(* Logix 5000 project; controller PLC vendor 1 type 14 code 155 rev 30.14; software revision 30.01; part 3 of 4 *)
(* tags used below, declared in another part *)
   Alarm_Word_Current : DINT[3];
   Bridge_Timer_Gearing_Delay : TIMER;
   Bridge_Timer_Gearing_Delay_DN_OS : BOOL;
   Depositor : Depositor_R2b;
   Encoder_Conveyor : AXIS_CIP_DRIVE;
   FORCE_GO_SIGNAL : BOOL;
   Forces : Forces_R2b;
   homing_timeout : TIMER;
   IO : IO_R2a;
   MV_conveyor_stopped : BOOL;
   MV_Encoder_Stop_Value : REAL;
   mv_index_counter : COUNTER;
   MV_indexes : DINT;
   MV_total_indexes : COUNTER;
   OS : INT[10];
   Recipe_Setpoints_DINT : DINT[23,20];
   Sequencer_Auto : Sequencer_R2a;
   Sequencer_Home : Sequencer_R2a;
   Servo_Bridge_Shift : AXIS_CIP_DRIVE;
   Servo_MC_Bridge_Shift : Axis_MC_R3b;
   System : System_R2e;
   Test_Bits : BOOL[32];
   Timers : TIMER[20];   // x
(* MainProgram, continued *)

ROUTINE File_012_Digital_Outputs   (* ladder *)
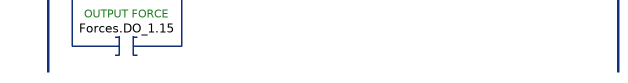
   // DIGITAL OUTPUT MAPPING
   0: [[XIC(IO.DO_1.0) ,XIC(Forces.DO_1.0) ] OTE(Local:1:O.Data.0) ,[XIC(IO.DO_1.1) ,XIC(Forces.DO_1.1) ] OTE(Local:1:O.Data.1) ,[XIC(IO.DO_1.2) ,XIC(Forces.DO_1.2) ] OTE(Local:1:O.Data.2) ,[XIC(IO.DO_1.3) ,XIC(Forces.DO_1.3) ] OTE(Local:1:O.Data.3) ,[XIC(IO.DO_1.4) ,XIC(Forces.DO_1.4) ] OTE(Local:1:O.Data.4) ,[XIC(IO.DO_1.5) ,XIC(Forces.DO_1.5) ] OTE(Local:1:O.Data.5) ,[XIC(IO.DO_1.6) ,XIC(Forces.DO_1.6) ] OTE(Local:1:O.Data.6) ,[XIC(IO.DO_1.7) ,XIC(Forces.DO_1.7) ] OTE(Local:1:O.Data.7) ,[XIC(IO.DO_1.8) ,XIC(Forces.DO_1.8) ] OTE(Local:1:O.Data.8) ,[XIC(IO.DO_1.9) ,XIC(Forces.DO_1.9) ] OTE(Local:1:O.Data.9) ,[XIC(IO.DO_1.10) ,XIC(Forces.DO_1.10) ] OTE(Local:1:O.Data.10) ,[XIC(IO.DO_1.11) ,XIC(Forces.DO_1.11) ] OTE(Local:1:O.Data.11) ,[XIC(IO.DO_1.12) ,XIC(Forces.DO_1.12) ] OTE(Local:1:O.Data.12) ,[XIC(IO.DO_1.13) ,XIC(Forces.DO_1.13) ] OTE(Local:1:O.Data.13) ,[XIC(IO.DO_1.14) ,XIC(Forces.DO_1.14) ] OTE(Local:1:O.Data.14) ,[XIC(IO.DO_1.15) ,XIC(Forces.DO_1.15) ] OTE(Local:1:O.Data.15) ];
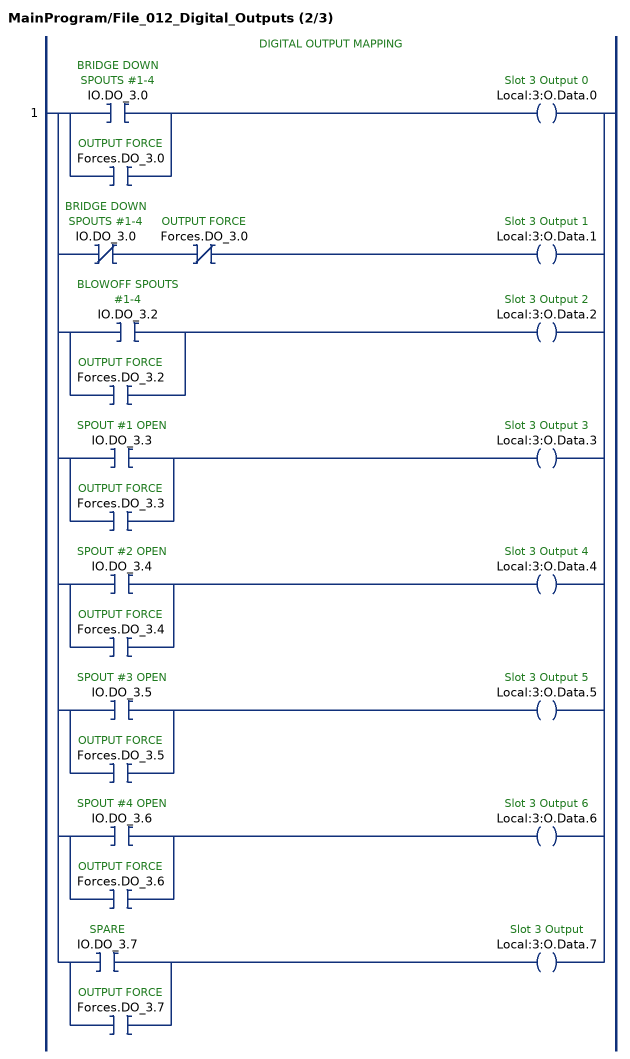
   // DIGITAL OUTPUT MAPPING
   1: [[XIC(IO.DO_3.0) ,XIC(Forces.DO_3.0) ] OTE(Local:3:O.Data.0) ,XIO(IO.DO_3.0) XIO(Forces.DO_3.0) OTE(Local:3:O.Data.1) ,[XIC(IO.DO_3.2) ,XIC(Forces.DO_3.2) ] OTE(Local:3:O.Data.2) ,[XIC(IO.DO_3.3) ,XIC(Forces.DO_3.3) ] OTE(Local:3:O.Data.3) ,[XIC(IO.DO_3.4) ,XIC(Forces.DO_3.4) ] OTE(Local:3:O.Data.4) ,[XIC(IO.DO_3.5) ,XIC(Forces.DO_3.5) ] OTE(Local:3:O.Data.5) ,[XIC(IO.DO_3.6) ,XIC(Forces.DO_3.6) ] OTE(Local:3:O.Data.6) ,[XIC(IO.DO_3.7) ,XIC(Forces.DO_3.7) ] OTE(Local:3:O.Data.7) ];
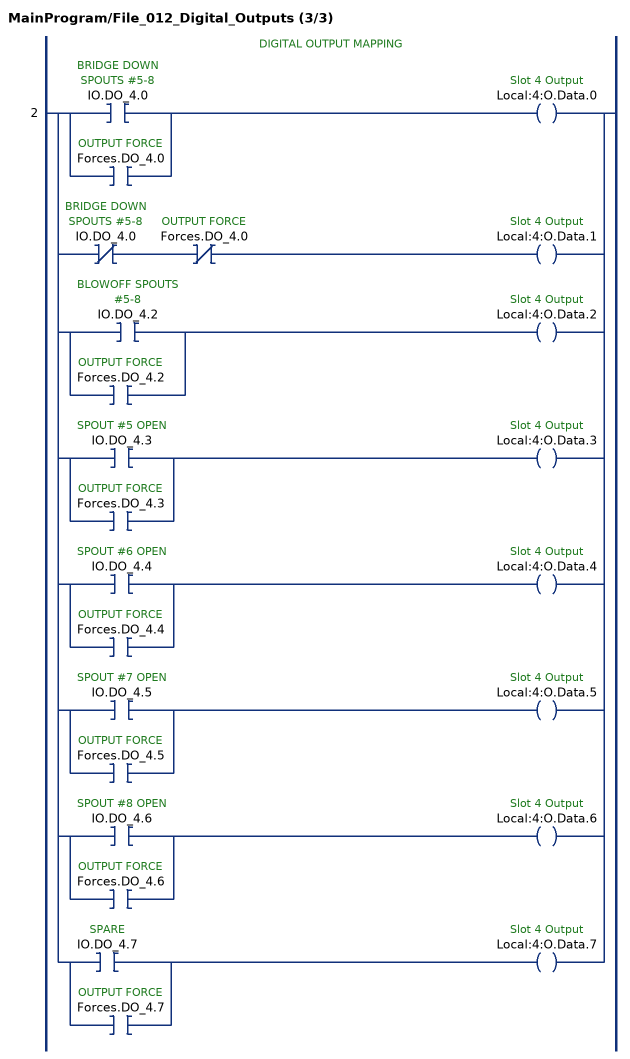
   // DIGITAL OUTPUT MAPPING
   2: [[XIC(IO.DO_4.0) ,XIC(Forces.DO_4.0) ] OTE(Local:4:O.Data.0) ,XIO(IO.DO_4.0) XIO(Forces.DO_4.0) OTE(Local:4:O.Data.1) ,[XIC(IO.DO_4.2) ,XIC(Forces.DO_4.2) ] OTE(Local:4:O.Data.2) ,[XIC(IO.DO_4.3) ,XIC(Forces.DO_4.3) ] OTE(Local:4:O.Data.3) ,[XIC(IO.DO_4.4) ,XIC(Forces.DO_4.4) ] OTE(Local:4:O.Data.4) ,[XIC(IO.DO_4.5) ,XIC(Forces.DO_4.5) ] OTE(Local:4:O.Data.5) ,[XIC(IO.DO_4.6) ,XIC(Forces.DO_4.6) ] OTE(Local:4:O.Data.6) ,[XIC(IO.DO_4.7) ,XIC(Forces.DO_4.7) ] OTE(Local:4:O.Data.7) ];
END_ROUTINE

ROUTINE File_030_Sequencer_Homing   (* ladder *)
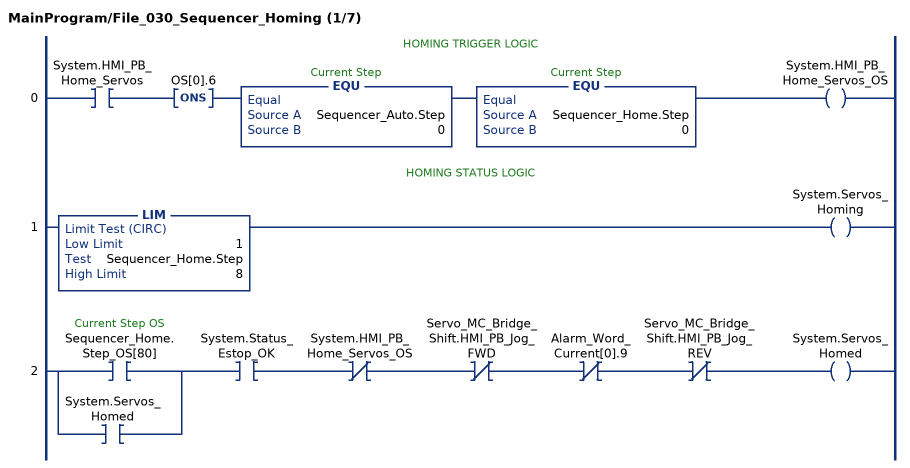
   // HOMING TRIGGER LOGIC
   0: XIC(System.HMI_PB_Home_Servos)ONS(OS[0].6)EQU(Sequencer_Auto.Step,0)EQU(Sequencer_Home.Step,0)OTE(System.HMI_PB_Home_Servos_OS);
   // HOMING STATUS LOGIC
   1: LIM(1,Sequencer_Home.Step,8)OTE(System.Servos_Homing);
   2: [XIC(Sequencer_Home.Step_OS[80]) ,XIC(System.Servos_Homed) ]XIC(System.Status_Estop_OK)XIO(System.HMI_PB_Home_Servos_OS)XIO(Servo_MC_Bridge_Shift.HMI_PB_Jog_FWD)XIO(Alarm_Word_Current[0].9)XIO(Servo_MC_Bridge_Shift.HMI_PB_Jog_REV)OTE(System.Servos_Homed);
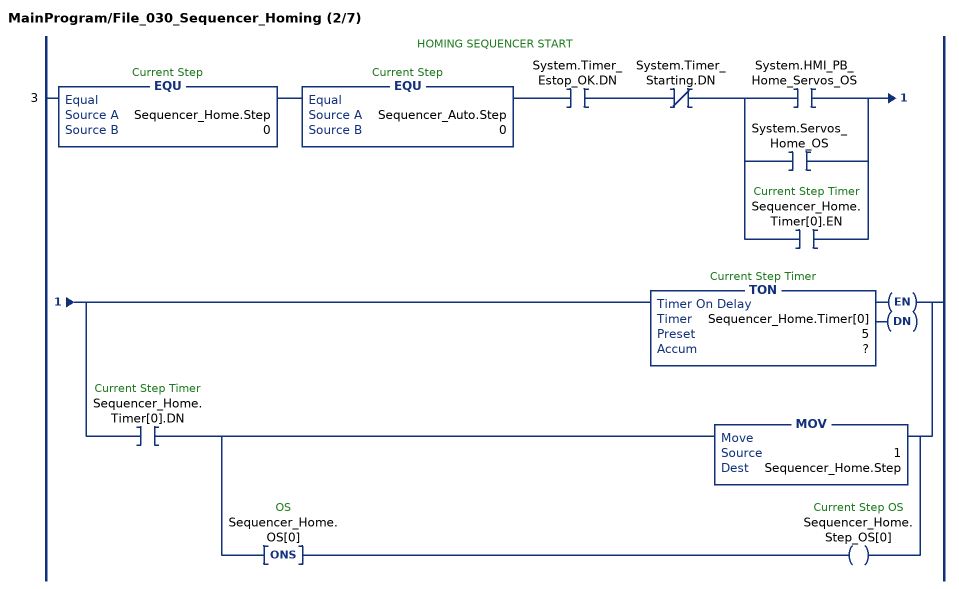
   // HOMING SEQUENCER START
   3: EQU(Sequencer_Home.Step,0)EQU(Sequencer_Auto.Step,0)XIC(System.Timer_Estop_OK.DN)XIO(System.Timer_Starting.DN)[XIC(System.HMI_PB_Home_Servos_OS) ,XIC(System.Servos_Home_OS) ,XIC(Sequencer_Home.Timer[0].EN) ][TON(Sequencer_Home.Timer[0],?,?) ,XIC(Sequencer_Home.Timer[0].DN) [MOV(1,Sequencer_Home.Step) ,ONS(Sequencer_Home.OS[0]) OTE(Sequencer_Home.Step_OS[0]) ] ];
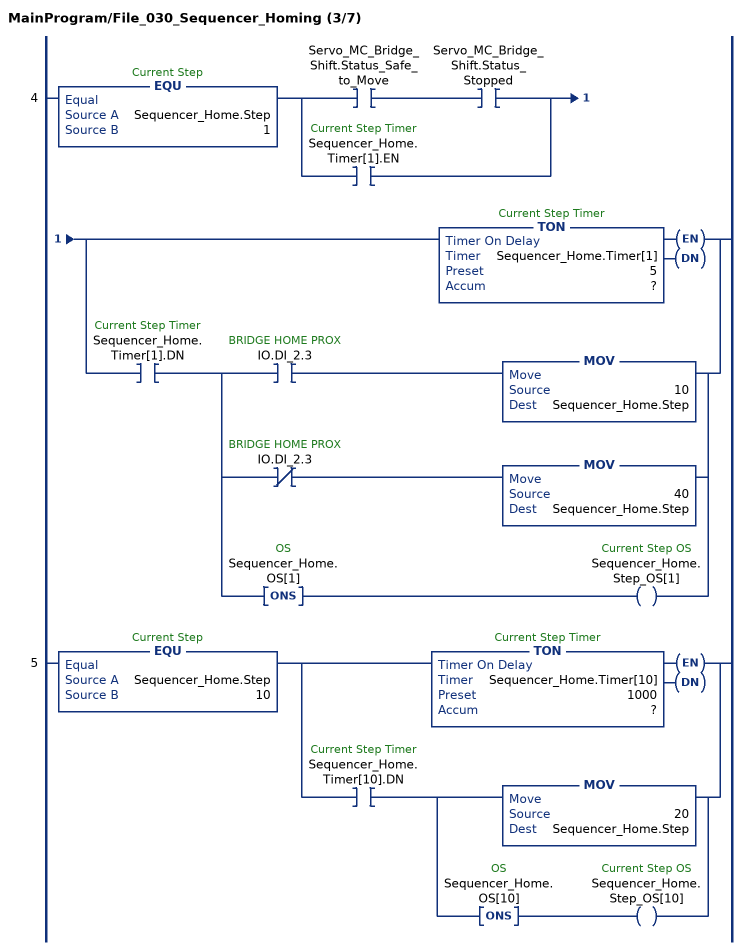
   4: EQU(Sequencer_Home.Step,1)[XIC(Servo_MC_Bridge_Shift.Status_Safe_to_Move) XIC(Servo_MC_Bridge_Shift.Status_Stopped) ,XIC(Sequencer_Home.Timer[1].EN) ][TON(Sequencer_Home.Timer[1],?,?) ,XIC(Sequencer_Home.Timer[1].DN) [XIC(IO.DI_2.3) MOV(10,Sequencer_Home.Step) ,XIO(IO.DI_2.3) MOV(40,Sequencer_Home.Step) ,ONS(Sequencer_Home.OS[1]) OTE(Sequencer_Home.Step_OS[1]) ] ];
   5: EQU(Sequencer_Home.Step,10)[TON(Sequencer_Home.Timer[10],?,?) ,XIC(Sequencer_Home.Timer[10].DN) [MOV(20,Sequencer_Home.Step) ,ONS(Sequencer_Home.OS[10]) OTE(Sequencer_Home.Step_OS[10]) ] ];
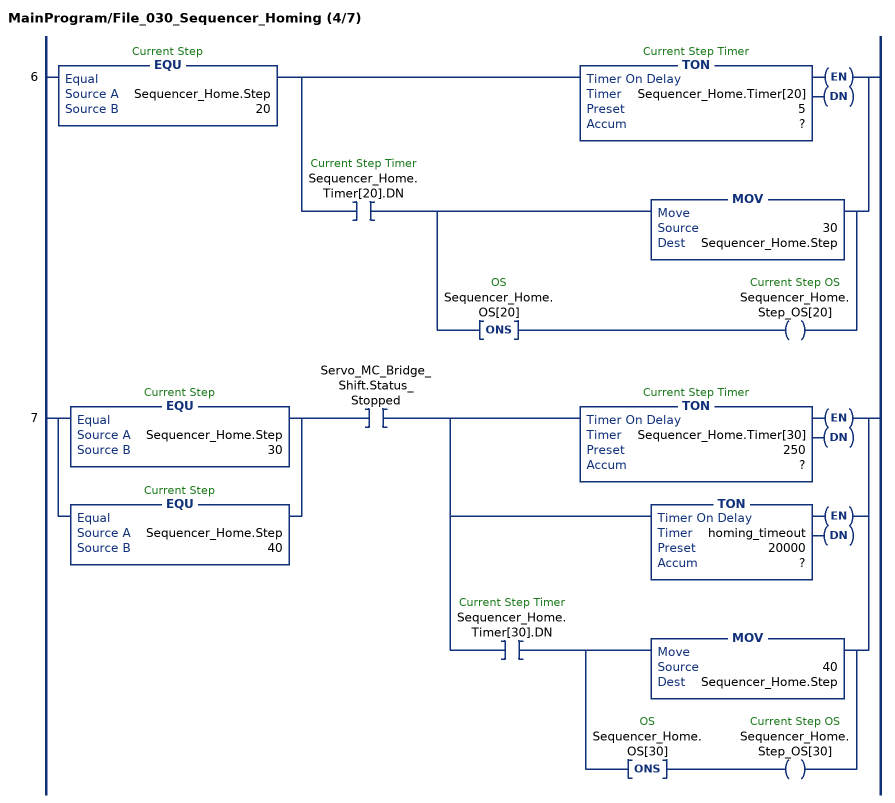
   6: EQU(Sequencer_Home.Step,20)[TON(Sequencer_Home.Timer[20],?,?) ,XIC(Sequencer_Home.Timer[20].DN) [MOV(30,Sequencer_Home.Step) ,ONS(Sequencer_Home.OS[20]) OTE(Sequencer_Home.Step_OS[20]) ] ];
   7: [EQU(Sequencer_Home.Step,30) ,EQU(Sequencer_Home.Step,40) ]XIC(Servo_MC_Bridge_Shift.Status_Stopped)[[TON(Sequencer_Home.Timer[30],?,?) ,TON(homing_timeout,?,?) ] ,XIC(Sequencer_Home.Timer[30].DN) [MOV(40,Sequencer_Home.Step) ,ONS(Sequencer_Home.OS[30]) OTE(Sequencer_Home.Step_OS[30]) ] ];
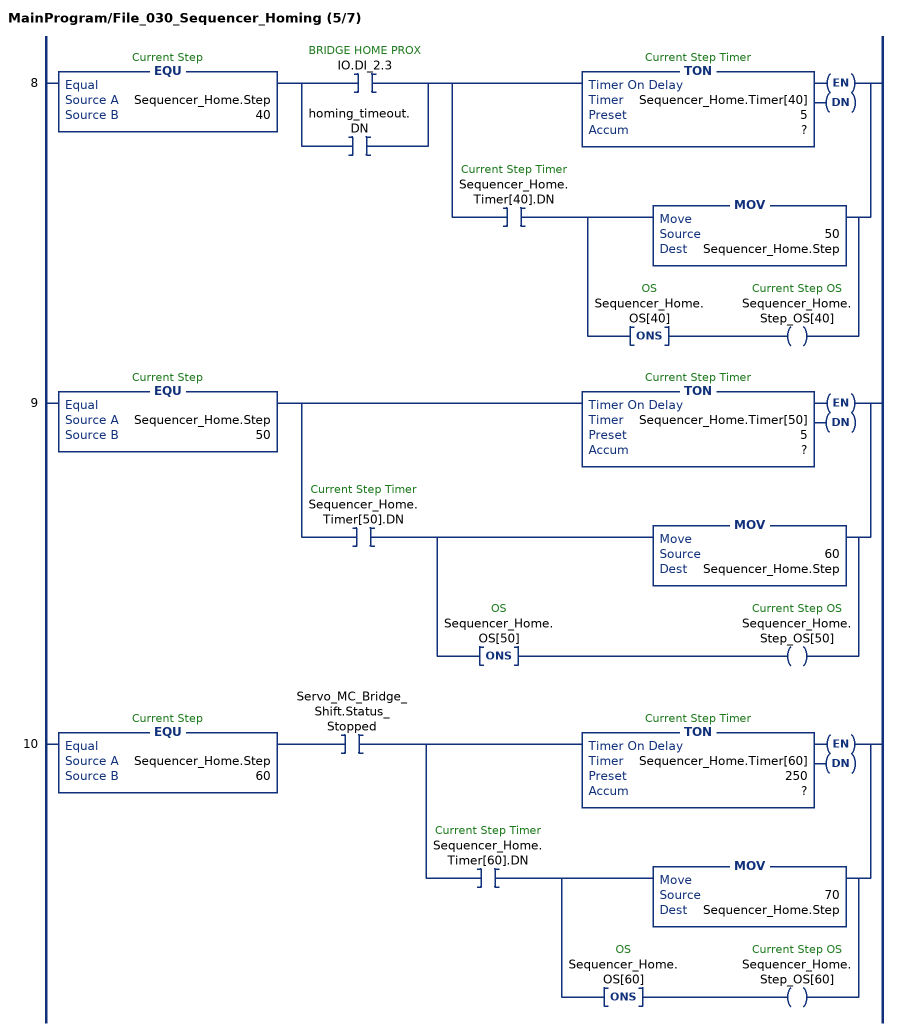
   8: EQU(Sequencer_Home.Step,40)[XIC(IO.DI_2.3) ,XIC(homing_timeout.DN) ][TON(Sequencer_Home.Timer[40],?,?) ,XIC(Sequencer_Home.Timer[40].DN) [MOV(50,Sequencer_Home.Step) ,ONS(Sequencer_Home.OS[40]) OTE(Sequencer_Home.Step_OS[40]) ] ];
   9: EQU(Sequencer_Home.Step,50)[TON(Sequencer_Home.Timer[50],?,?) ,XIC(Sequencer_Home.Timer[50].DN) [MOV(60,Sequencer_Home.Step) ,ONS(Sequencer_Home.OS[50]) OTE(Sequencer_Home.Step_OS[50]) ] ];
   10: EQU(Sequencer_Home.Step,60)XIC(Servo_MC_Bridge_Shift.Status_Stopped)[TON(Sequencer_Home.Timer[60],?,?) ,XIC(Sequencer_Home.Timer[60].DN) [MOV(70,Sequencer_Home.Step) ,ONS(Sequencer_Home.OS[60]) OTE(Sequencer_Home.Step_OS[60]) ] ];
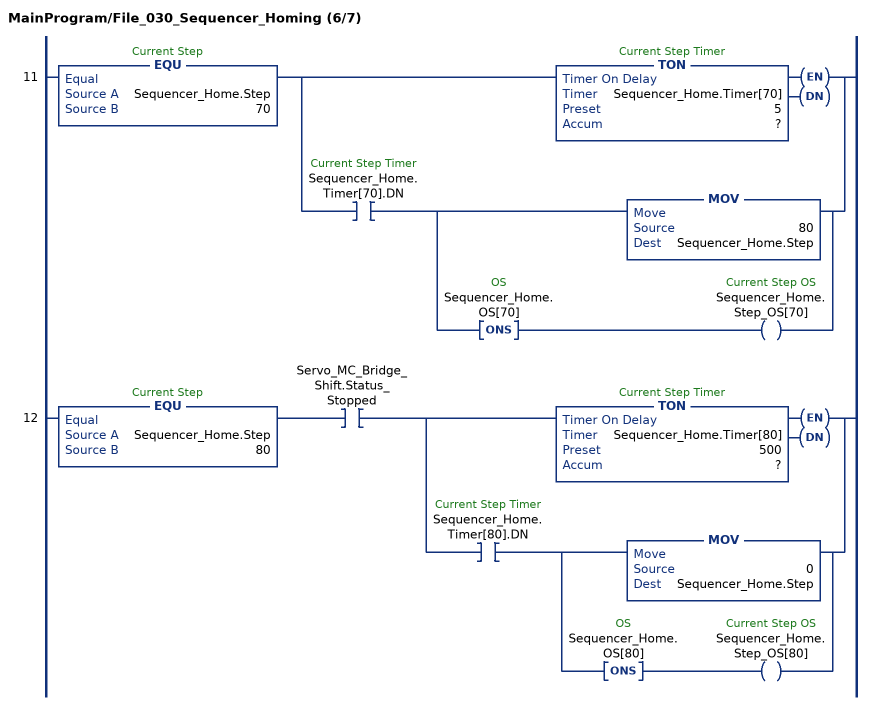
   11: EQU(Sequencer_Home.Step,70)[TON(Sequencer_Home.Timer[70],?,?) ,XIC(Sequencer_Home.Timer[70].DN) [MOV(80,Sequencer_Home.Step) ,ONS(Sequencer_Home.OS[70]) OTE(Sequencer_Home.Step_OS[70]) ] ];
   12: EQU(Sequencer_Home.Step,80)XIC(Servo_MC_Bridge_Shift.Status_Stopped)[TON(Sequencer_Home.Timer[80],?,?) ,XIC(Sequencer_Home.Timer[80].DN) [MOV(0,Sequencer_Home.Step) ,ONS(Sequencer_Home.OS[80]) OTE(Sequencer_Home.Step_OS[80]) ] ];
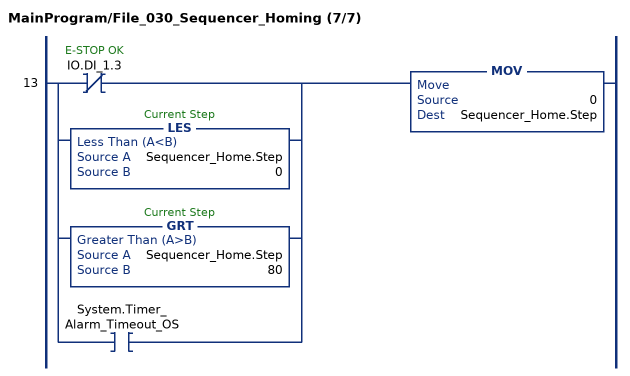
   13: [XIO(IO.DI_1.3) ,LES(Sequencer_Home.Step,0) ,GRT(Sequencer_Home.Step,80) ,XIC(System.Timer_Alarm_Timeout_OS) ]MOV(0,Sequencer_Home.Step);
END_ROUTINE

ROUTINE File_040_Sequencer_Auto   (* ladder *)
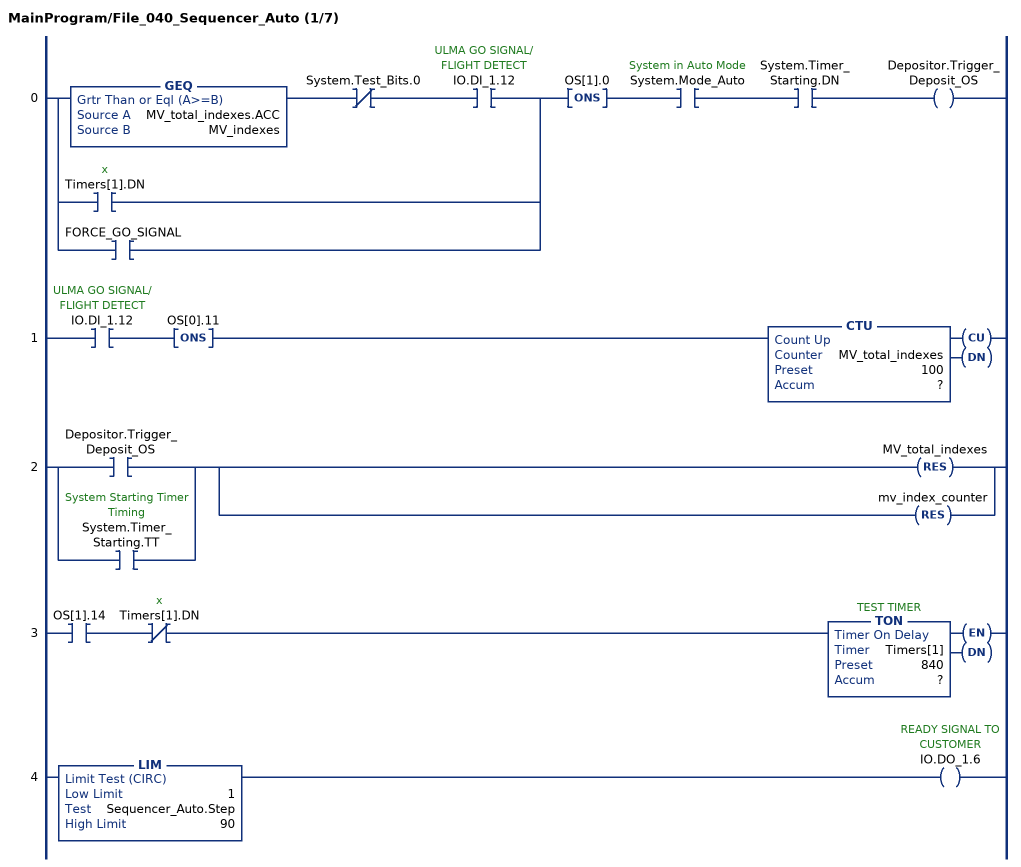
   0: [GEQ(MV_total_indexes.ACC,MV_indexes) XIO(System.Test_Bits.0) XIC(IO.DI_1.12) ,XIC(Timers[1].DN) ,XIC(FORCE_GO_SIGNAL) ]ONS(OS[1].0)XIC(System.Mode_Auto)XIC(System.Timer_Starting.DN)OTE(Depositor.Trigger_Deposit_OS);
   1: XIC(IO.DI_1.12)ONS(OS[0].11)CTU(MV_total_indexes,?,?);
   2: [XIC(Depositor.Trigger_Deposit_OS) ,XIC(System.Timer_Starting.TT) ][RES(MV_total_indexes) ,RES(mv_index_counter) ];
   3: XIC(OS[1].14)XIO(Timers[1].DN)TON(Timers[1],?,?);
   4: LIM(1,Sequencer_Auto.Step,90)OTE(IO.DO_1.6);
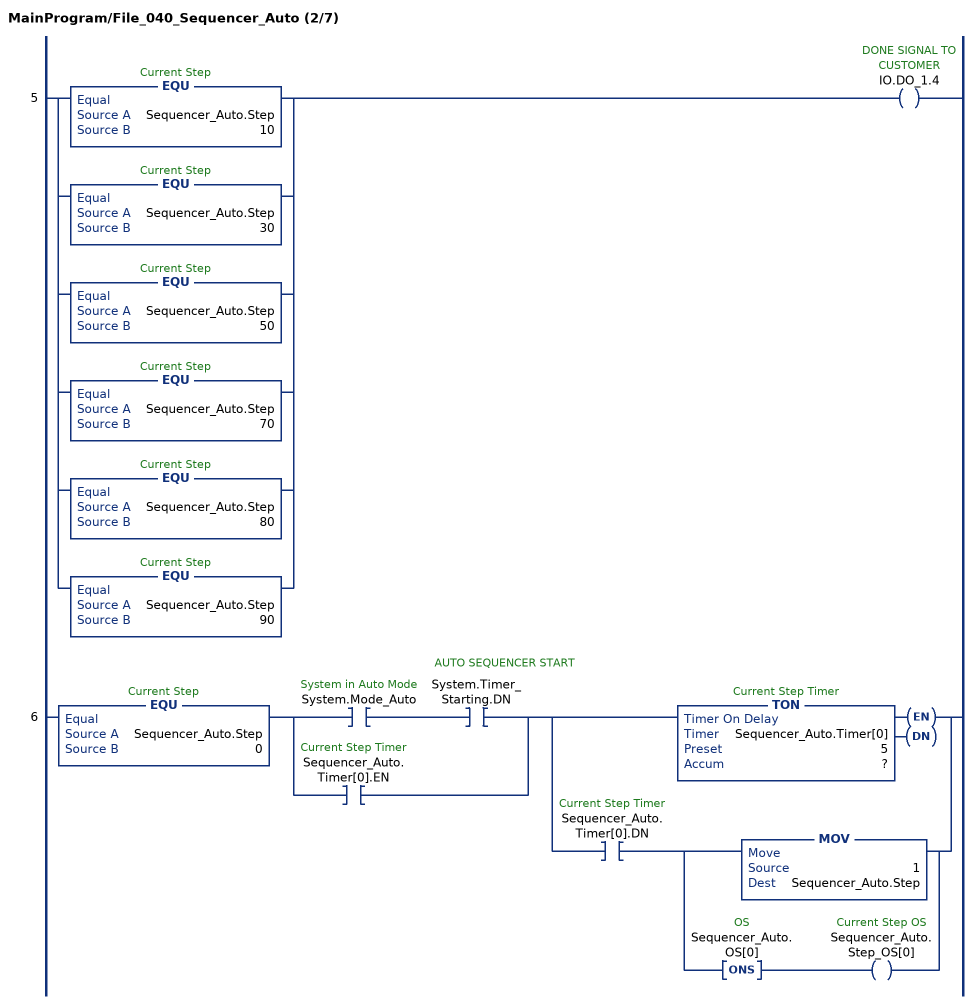
   5: [EQU(Sequencer_Auto.Step,10) ,EQU(Sequencer_Auto.Step,30) ,EQU(Sequencer_Auto.Step,50) ,EQU(Sequencer_Auto.Step,70) ,EQU(Sequencer_Auto.Step,80) ,EQU(Sequencer_Auto.Step,90) ]OTE(IO.DO_1.4);
   // AUTO SEQUENCER START
   6: EQU(Sequencer_Auto.Step,0)[XIC(System.Mode_Auto) XIC(System.Timer_Starting.DN) ,XIC(Sequencer_Auto.Timer[0].EN) ][TON(Sequencer_Auto.Timer[0],?,?) ,XIC(Sequencer_Auto.Timer[0].DN) [MOV(1,Sequencer_Auto.Step) ,ONS(Sequencer_Auto.OS[0]) OTE(Sequencer_Auto.Step_OS[0]) ] ];
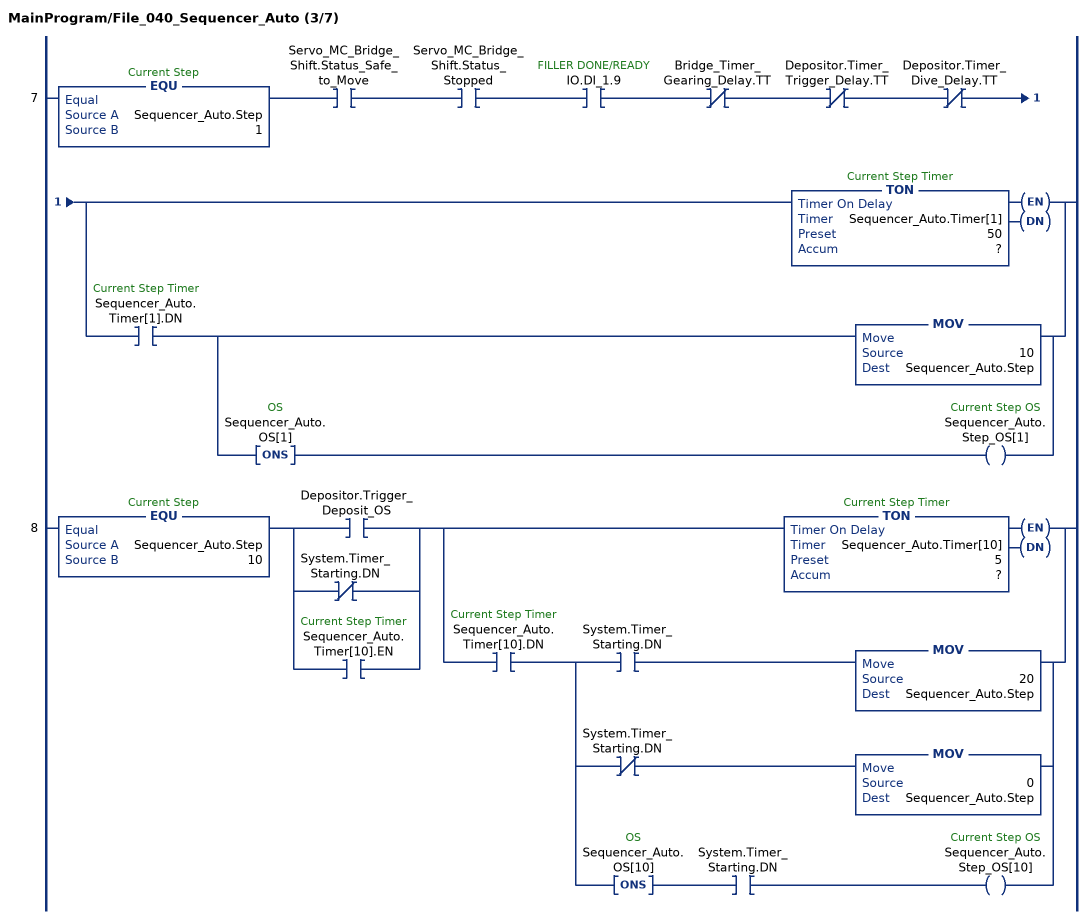
   7: EQU(Sequencer_Auto.Step,1)XIC(Servo_MC_Bridge_Shift.Status_Safe_to_Move)XIC(Servo_MC_Bridge_Shift.Status_Stopped)XIC(IO.DI_1.9)XIO(Bridge_Timer_Gearing_Delay.TT)XIO(Depositor.Timer_Trigger_Delay.TT)XIO(Depositor.Timer_Dive_Delay.TT)[TON(Sequencer_Auto.Timer[1],?,?) ,XIC(Sequencer_Auto.Timer[1].DN) [MOV(10,Sequencer_Auto.Step) ,ONS(Sequencer_Auto.OS[1]) OTE(Sequencer_Auto.Step_OS[1]) ] ];
   8: EQU(Sequencer_Auto.Step,10)[XIC(Depositor.Trigger_Deposit_OS) ,XIO(System.Timer_Starting.DN) ,XIC(Sequencer_Auto.Timer[10].EN) ][TON(Sequencer_Auto.Timer[10],?,?) ,XIC(Sequencer_Auto.Timer[10].DN) [XIC(System.Timer_Starting.DN) MOV(20,Sequencer_Auto.Step) ,XIO(System.Timer_Starting.DN) MOV(0,Sequencer_Auto.Step) ,ONS(Sequencer_Auto.OS[10]) XIC(System.Timer_Starting.DN) OTE(Sequencer_Auto.Step_OS[10]) ] ];
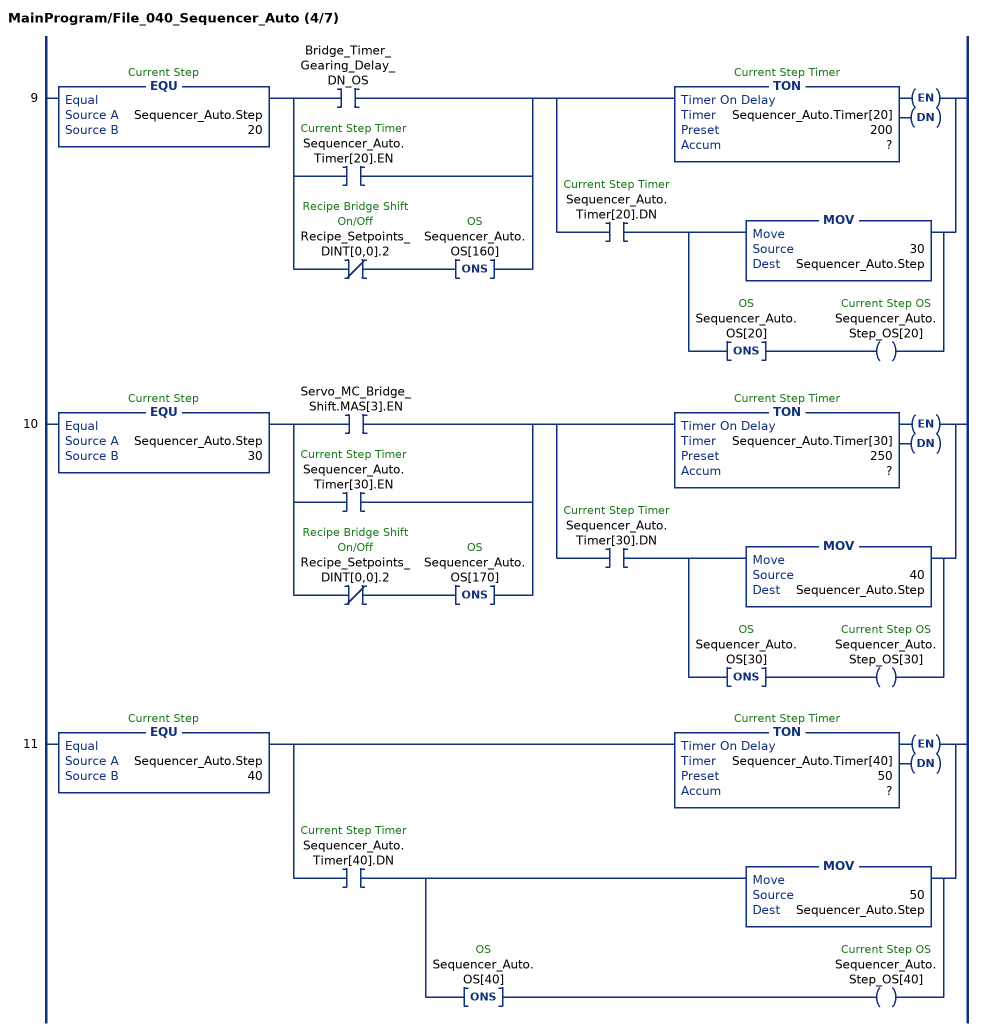
   9: EQU(Sequencer_Auto.Step,20)[XIC(Bridge_Timer_Gearing_Delay_DN_OS) ,XIC(Sequencer_Auto.Timer[20].EN) ,XIO(Recipe_Setpoints_DINT[0,0].2) ONS(Sequencer_Auto.OS[160]) ][TON(Sequencer_Auto.Timer[20],?,?) ,XIC(Sequencer_Auto.Timer[20].DN) [MOV(30,Sequencer_Auto.Step) ,ONS(Sequencer_Auto.OS[20]) OTE(Sequencer_Auto.Step_OS[20]) ] ];
   10: EQU(Sequencer_Auto.Step,30)[XIC(Servo_MC_Bridge_Shift.MAS[3].EN) ,XIC(Sequencer_Auto.Timer[30].EN) ,XIO(Recipe_Setpoints_DINT[0,0].2) ONS(Sequencer_Auto.OS[170]) ][TON(Sequencer_Auto.Timer[30],?,?) ,XIC(Sequencer_Auto.Timer[30].DN) [MOV(40,Sequencer_Auto.Step) ,ONS(Sequencer_Auto.OS[30]) OTE(Sequencer_Auto.Step_OS[30]) ] ];
   11: EQU(Sequencer_Auto.Step,40)[TON(Sequencer_Auto.Timer[40],?,?) ,XIC(Sequencer_Auto.Timer[40].DN) [MOV(50,Sequencer_Auto.Step) ,ONS(Sequencer_Auto.OS[40]) OTE(Sequencer_Auto.Step_OS[40]) ] ];
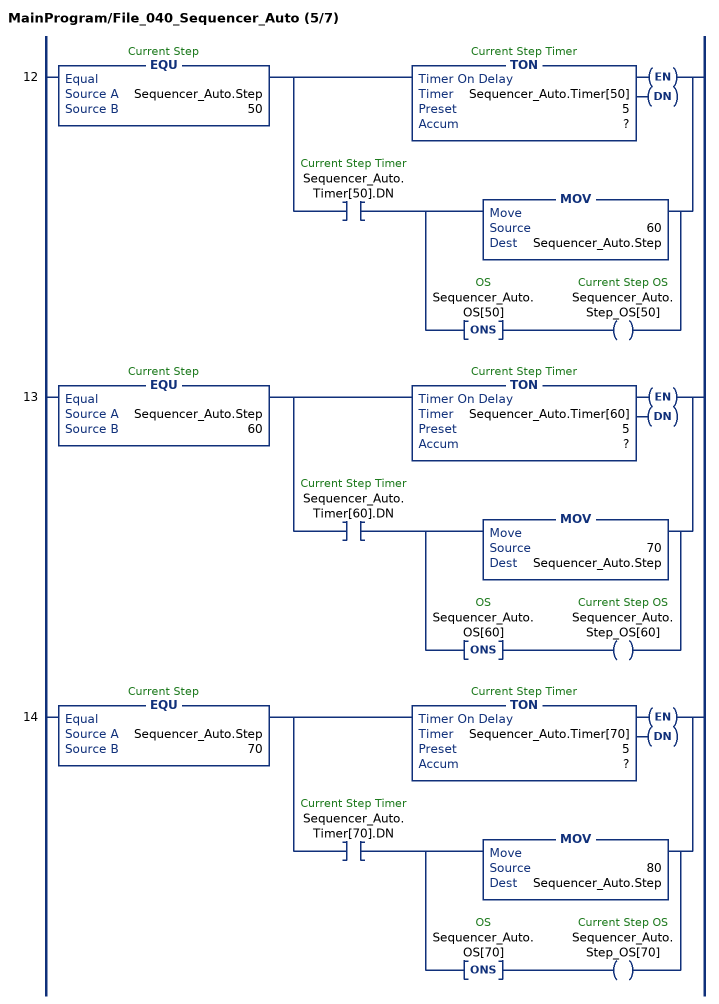
   12: EQU(Sequencer_Auto.Step,50)[TON(Sequencer_Auto.Timer[50],?,?) ,XIC(Sequencer_Auto.Timer[50].DN) [MOV(60,Sequencer_Auto.Step) ,ONS(Sequencer_Auto.OS[50]) OTE(Sequencer_Auto.Step_OS[50]) ] ];
   13: EQU(Sequencer_Auto.Step,60)[TON(Sequencer_Auto.Timer[60],?,?) ,XIC(Sequencer_Auto.Timer[60].DN) [MOV(70,Sequencer_Auto.Step) ,ONS(Sequencer_Auto.OS[60]) OTE(Sequencer_Auto.Step_OS[60]) ] ];
   14: EQU(Sequencer_Auto.Step,70)[TON(Sequencer_Auto.Timer[70],?,?) ,XIC(Sequencer_Auto.Timer[70].DN) [MOV(80,Sequencer_Auto.Step) ,ONS(Sequencer_Auto.OS[70]) OTE(Sequencer_Auto.Step_OS[70]) ] ];
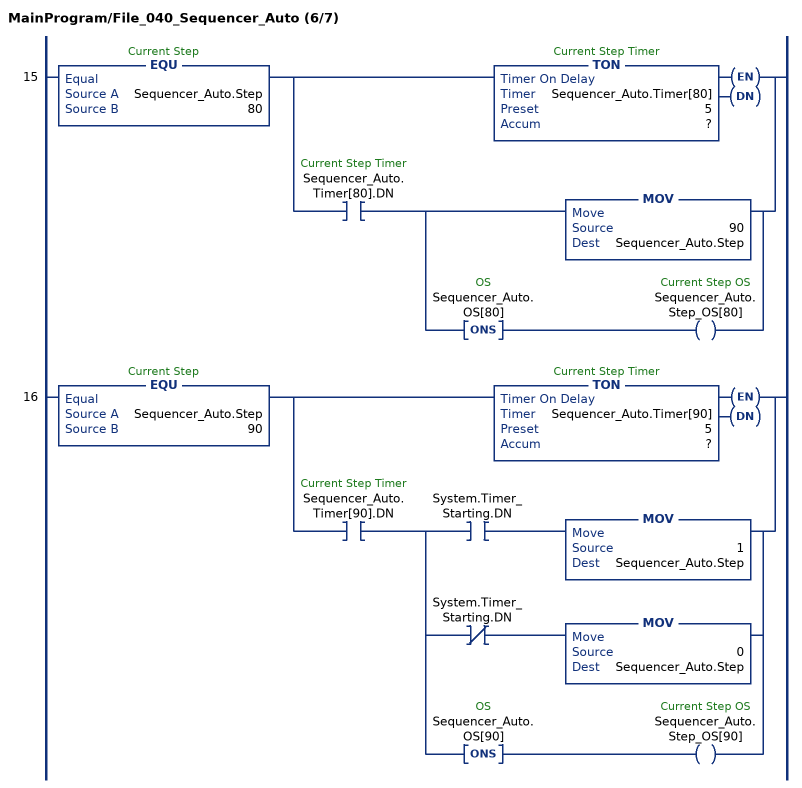
   15: EQU(Sequencer_Auto.Step,80)[TON(Sequencer_Auto.Timer[80],?,?) ,XIC(Sequencer_Auto.Timer[80].DN) [MOV(90,Sequencer_Auto.Step) ,ONS(Sequencer_Auto.OS[80]) OTE(Sequencer_Auto.Step_OS[80]) ] ];
   16: EQU(Sequencer_Auto.Step,90)[TON(Sequencer_Auto.Timer[90],?,?) ,XIC(Sequencer_Auto.Timer[90].DN) [XIC(System.Timer_Starting.DN) MOV(1,Sequencer_Auto.Step) ,XIO(System.Timer_Starting.DN) MOV(0,Sequencer_Auto.Step) ,ONS(Sequencer_Auto.OS[90]) OTE(Sequencer_Auto.Step_OS[90]) ] ];
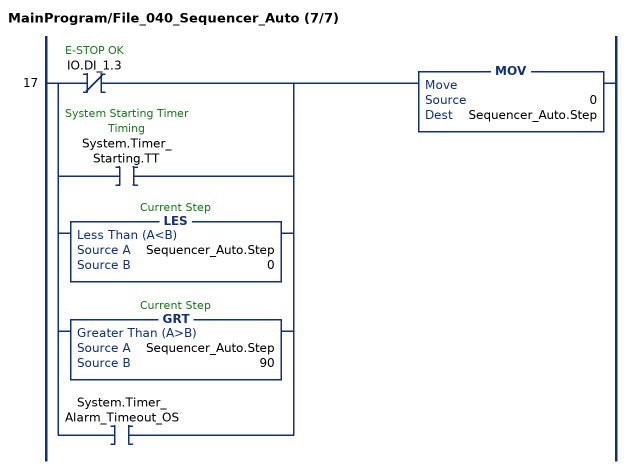
   17: [XIO(IO.DI_1.3) ,XIC(System.Timer_Starting.TT) ,LES(Sequencer_Auto.Step,0) ,GRT(Sequencer_Auto.Step,90) ,XIC(System.Timer_Alarm_Timeout_OS) ]MOV(0,Sequencer_Auto.Step);
END_ROUTINE

ROUTINE File_100_Servo_Bridge   (* ladder *)
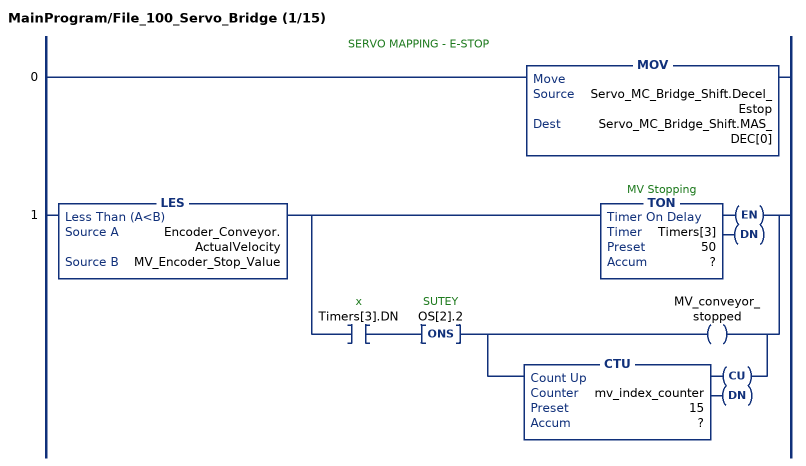
   // SERVO MAPPING - E-STOP
   0: MOV(Servo_MC_Bridge_Shift.Decel_Estop,Servo_MC_Bridge_Shift.MAS_DEC[0]);
   1: LES(Encoder_Conveyor.ActualVelocity,MV_Encoder_Stop_Value)[TON(Timers[3],?,?) ,XIC(Timers[3].DN) ONS(OS[2].2) [OTE(MV_conveyor_stopped) ,CTU(mv_index_counter,?,?) ] ];
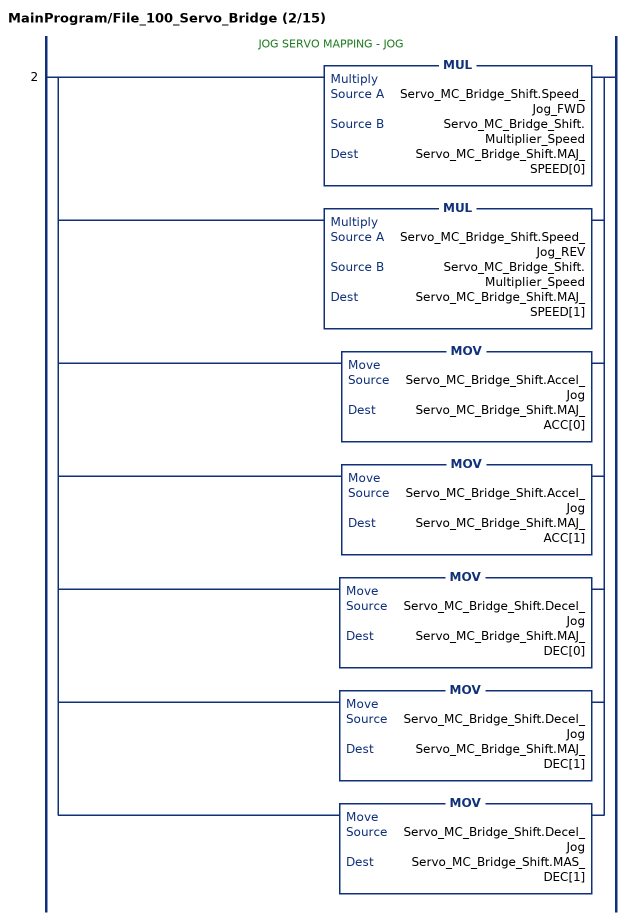
   // JOG SERVO MAPPING - JOG
   2: [MUL(Servo_MC_Bridge_Shift.Speed_Jog_FWD,Servo_MC_Bridge_Shift.Multiplier_Speed,Servo_MC_Bridge_Shift.MAJ_SPEED[0]) ,MUL(Servo_MC_Bridge_Shift.Speed_Jog_REV,Servo_MC_Bridge_Shift.Multiplier_Speed,Servo_MC_Bridge_Shift.MAJ_SPEED[1]) ,MOV(Servo_MC_Bridge_Shift.Accel_Jog,Servo_MC_Bridge_Shift.MAJ_ACC[0]) ,MOV(Servo_MC_Bridge_Shift.Accel_Jog,Servo_MC_Bridge_Shift.MAJ_ACC[1]) ,MOV(Servo_MC_Bridge_Shift.Decel_Jog,Servo_MC_Bridge_Shift.MAJ_DEC[0]) ,MOV(Servo_MC_Bridge_Shift.Decel_Jog,Servo_MC_Bridge_Shift.MAJ_DEC[1]) ,MOV(Servo_MC_Bridge_Shift.Decel_Jog,Servo_MC_Bridge_Shift.MAS_DEC[1]) ];
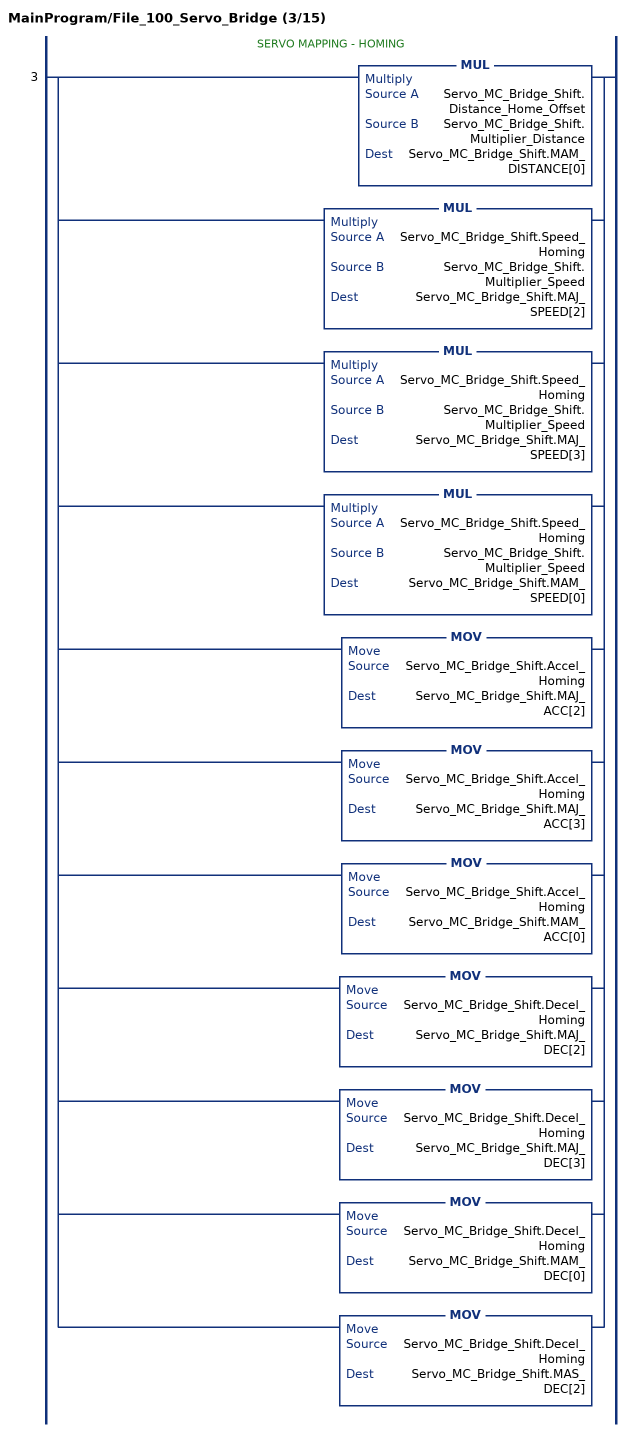
   // SERVO MAPPING - HOMING
   3: [MUL(Servo_MC_Bridge_Shift.Distance_Home_Offset,Servo_MC_Bridge_Shift.Multiplier_Distance,Servo_MC_Bridge_Shift.MAM_DISTANCE[0]) ,MUL(Servo_MC_Bridge_Shift.Speed_Homing,Servo_MC_Bridge_Shift.Multiplier_Speed,Servo_MC_Bridge_Shift.MAJ_SPEED[2]) ,MUL(Servo_MC_Bridge_Shift.Speed_Homing,Servo_MC_Bridge_Shift.Multiplier_Speed,Servo_MC_Bridge_Shift.MAJ_SPEED[3]) ,MUL(Servo_MC_Bridge_Shift.Speed_Homing,Servo_MC_Bridge_Shift.Multiplier_Speed,Servo_MC_Bridge_Shift.MAM_SPEED[0]) ,MOV(Servo_MC_Bridge_Shift.Accel_Homing,Servo_MC_Bridge_Shift.MAJ_ACC[2]) ,MOV(Servo_MC_Bridge_Shift.Accel_Homing,Servo_MC_Bridge_Shift.MAJ_ACC[3]) ,MOV(Servo_MC_Bridge_Shift.Accel_Homing,Servo_MC_Bridge_Shift.MAM_ACC[0]) ,MOV(Servo_MC_Bridge_Shift.Decel_Homing,Servo_MC_Bridge_Shift.MAJ_DEC[2]) ,MOV(Servo_MC_Bridge_Shift.Decel_Homing,Servo_MC_Bridge_Shift.MAJ_DEC[3]) ,MOV(Servo_MC_Bridge_Shift.Decel_Homing,Servo_MC_Bridge_Shift.MAM_DEC[0]) ,MOV(Servo_MC_Bridge_Shift.Decel_Homing,Servo_MC_Bridge_Shift.MAS_DEC[2]) ];
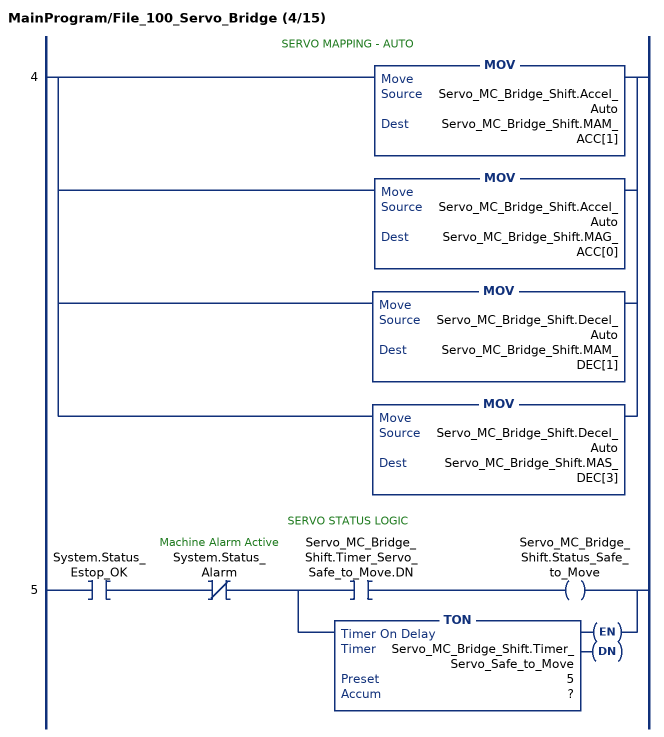
   // SERVO MAPPING - AUTO
   4: [MOV(Servo_MC_Bridge_Shift.Accel_Auto,Servo_MC_Bridge_Shift.MAM_ACC[1]) ,MOV(Servo_MC_Bridge_Shift.Accel_Auto,Servo_MC_Bridge_Shift.MAG_ACC[0]) ,MOV(Servo_MC_Bridge_Shift.Decel_Auto,Servo_MC_Bridge_Shift.MAM_DEC[1]) ,MOV(Servo_MC_Bridge_Shift.Decel_Auto,Servo_MC_Bridge_Shift.MAS_DEC[3]) ];
   // SERVO STATUS LOGIC
   5: XIC(System.Status_Estop_OK)XIO(System.Status_Alarm)[XIC(Servo_MC_Bridge_Shift.Timer_Servo_Safe_to_Move.DN) OTE(Servo_MC_Bridge_Shift.Status_Safe_to_Move) ,TON(Servo_MC_Bridge_Shift.Timer_Servo_Safe_to_Move,?,?) ];
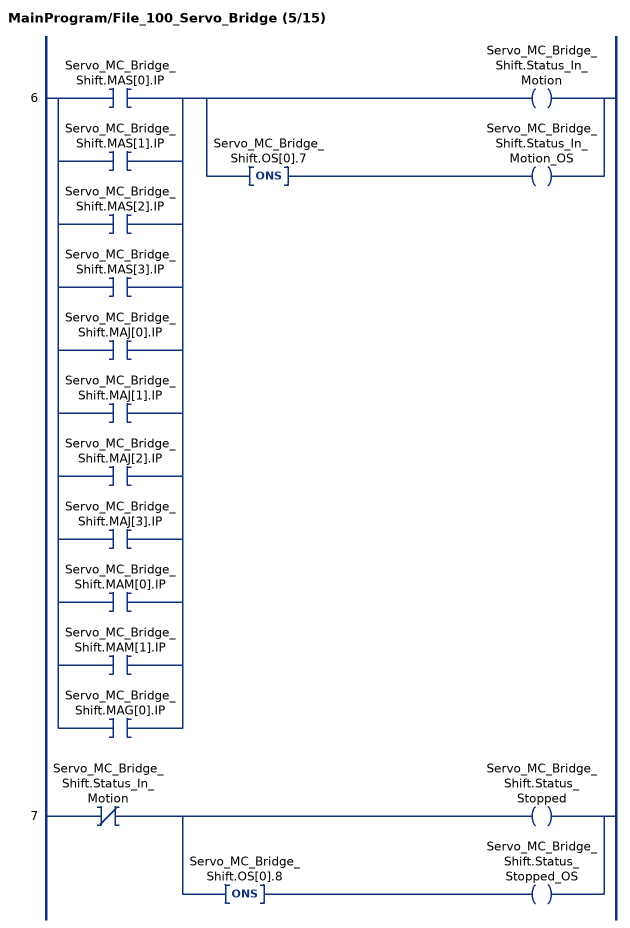
   6: [XIC(Servo_MC_Bridge_Shift.MAS[0].IP) ,XIC(Servo_MC_Bridge_Shift.MAS[1].IP) ,XIC(Servo_MC_Bridge_Shift.MAS[2].IP) ,XIC(Servo_MC_Bridge_Shift.MAS[3].IP) ,XIC(Servo_MC_Bridge_Shift.MAJ[0].IP) ,XIC(Servo_MC_Bridge_Shift.MAJ[1].IP) ,XIC(Servo_MC_Bridge_Shift.MAJ[2].IP) ,XIC(Servo_MC_Bridge_Shift.MAJ[3].IP) ,XIC(Servo_MC_Bridge_Shift.MAM[0].IP) ,XIC(Servo_MC_Bridge_Shift.MAM[1].IP) ,XIC(Servo_MC_Bridge_Shift.MAG[0].IP) ][OTE(Servo_MC_Bridge_Shift.Status_In_Motion) ,ONS(Servo_MC_Bridge_Shift.OS[0].7) OTE(Servo_MC_Bridge_Shift.Status_In_Motion_OS) ];
   7: XIO(Servo_MC_Bridge_Shift.Status_In_Motion)[OTE(Servo_MC_Bridge_Shift.Status_Stopped) ,ONS(Servo_MC_Bridge_Shift.OS[0].8) OTE(Servo_MC_Bridge_Shift.Status_Stopped_OS) ];
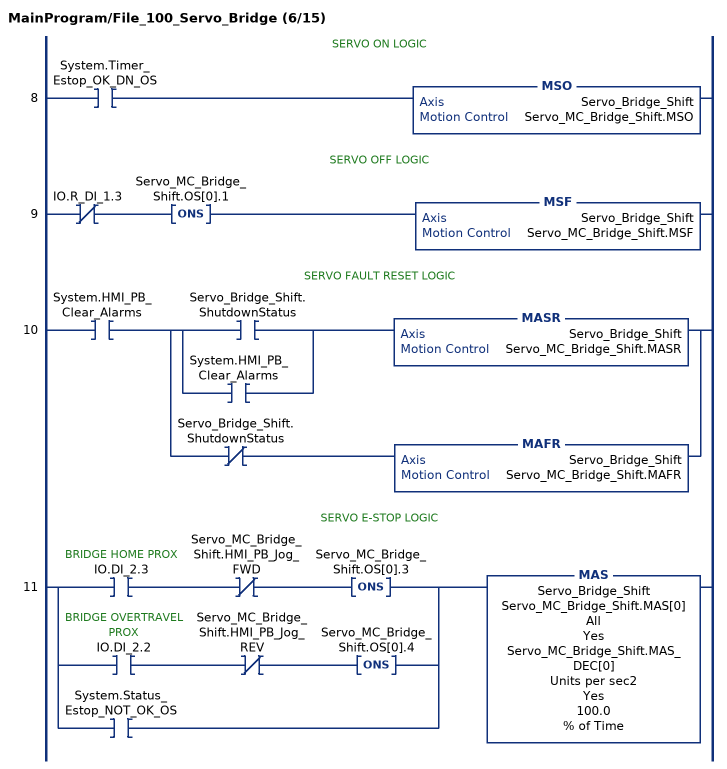
   // SERVO ON LOGIC
   8: XIC(System.Timer_Estop_OK_DN_OS)MSO(Servo_Bridge_Shift,Servo_MC_Bridge_Shift.MSO);
   // SERVO OFF LOGIC
   9: XIO(IO.R_DI_1.3)ONS(Servo_MC_Bridge_Shift.OS[0].1)MSF(Servo_Bridge_Shift,Servo_MC_Bridge_Shift.MSF);
   // SERVO FAULT RESET LOGIC
   10: XIC(System.HMI_PB_Clear_Alarms)[[XIC(Servo_Bridge_Shift.ShutdownStatus) ,XIC(System.HMI_PB_Clear_Alarms) ] MASR(Servo_Bridge_Shift,Servo_MC_Bridge_Shift.MASR) ,XIO(Servo_Bridge_Shift.ShutdownStatus) MAFR(Servo_Bridge_Shift,Servo_MC_Bridge_Shift.MAFR) ];
   // SERVO E-STOP LOGIC
   11: [XIC(IO.DI_2.3) XIO(Servo_MC_Bridge_Shift.HMI_PB_Jog_FWD) ONS(Servo_MC_Bridge_Shift.OS[0].3) ,XIC(IO.DI_2.2) XIO(Servo_MC_Bridge_Shift.HMI_PB_Jog_REV) ONS(Servo_MC_Bridge_Shift.OS[0].4) ,XIC(System.Status_Estop_NOT_OK_OS) ]MAS(Servo_Bridge_Shift,Servo_MC_Bridge_Shift.MAS[0],All,Yes,Servo_MC_Bridge_Shift.MAS_DEC[0],Units per sec2,Yes,100.0,% of Time);
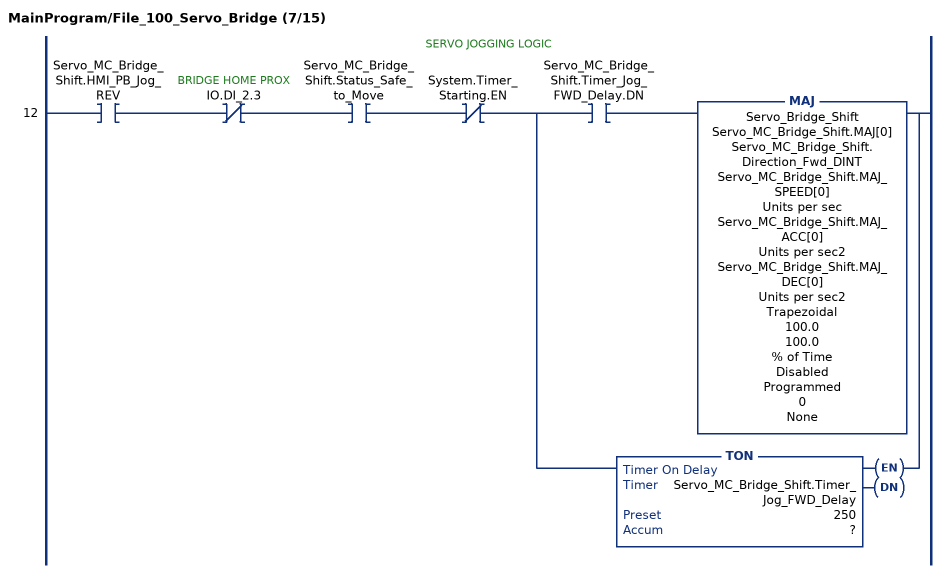
   // SERVO JOGGING LOGIC
   12: XIC(Servo_MC_Bridge_Shift.HMI_PB_Jog_REV)XIO(IO.DI_2.3)XIC(Servo_MC_Bridge_Shift.Status_Safe_to_Move)XIO(System.Timer_Starting.EN)[XIC(Servo_MC_Bridge_Shift.Timer_Jog_FWD_Delay.DN) MAJ(Servo_Bridge_Shift,Servo_MC_Bridge_Shift.MAJ[0],Servo_MC_Bridge_Shift.Direction_Fwd_DINT,Servo_MC_Bridge_Shift.MAJ_SPEED[0],Units per sec,Servo_MC_Bridge_Shift.MAJ_ACC[0],Units per sec2,Servo_MC_Bridge_Shift.MAJ_DEC[0],Units per sec2,Trapezoidal,100.0,100.0,% of Time,Disabled,Programmed,0,None) ,TON(Servo_MC_Bridge_Shift.Timer_Jog_FWD_Delay,?,?) ];
